(* PLC project  *)

CONFIGURATION AxisMR
END_CONFIGURATION
